FUNCTION_BLOCK WatchdogTimer
VAR_INPUT
END_VAR
VAR_OUTPUT
END_VAR
VAR
END_VAR

END_FUNCTION_BLOCK

(* stored: Version 1.1.0.1, ProductVersion 3.1.4024.6
   POU WatchdogTimer: Id {ea05dca4-2630-471a-814d-f1294ce390fd}, SpecialFunc None *)
